{attribute addProperty BoxType "EK1122-0000-0018"}
{attribute addProperty Id "Beckhoff_ER4xxxsub_EK1100EK1100_179A0949162A_0001_ER4174_0002_0016ER4174_253CF8AE15219A_0002_ER4174_0002_0019ER4174_253CF8AE15219A_0003_ER4374_0002_0018ER4374_D464211E19224A_0004_ER4374_0002_0019ER4374_D464211E19224"}
{attribute addProperty CRC "2433570836"}
{attribute addProperty SizeInBites "704"}
{attribute addProperty SizeInBytes "88"}
TYPE Beckhoff_ER4xxxEK1122_910D5814 EXTENDS EK1122_179A0949 :
STRUCT
	{attribute addProperty Name "Beckhoff_ER4xxxsub_EK1100"}
	Beckhoff_ER4xxxsub_EK1100 : EK1100_179A0949;
	{attribute addProperty Name "A_0001_ER4174_0002_0016"}
	A_0001_ER4174_0002_0016 : ER4174_253CF8AE;
	{attribute addProperty Name "A_0002_ER4174_0002_0019"}
	A_0002_ER4174_0002_0019 : ER4174_253CF8AE;
	{attribute addProperty Name "A_0003_ER4374_0002_0018"}
	A_0003_ER4374_0002_0018 : ER4374_D464211E;
	{attribute addProperty Name "A_0004_ER4374_0002_0019"}
	A_0004_ER4374_0002_0019 : ER4374_D464211E;
END_STRUCT
END_TYPE

(* stored: Version 1.2.0.0, ProductVersion 3.1.4024.9
   DUT Beckhoff_ER4xxxEK1122_910D5814: Id {4dd7d4be-548e-4e34-a9a7-a14544079751} *)
